// Implicitly generated code : DO NOT EDIT
FUNCTION CheckLRangeSigned : LINT
VAR_INPUT
	value, lower, upper: LINT;
END_VAR

{noflow}
IF (value < lower) THEN
	CheckLRangeSigned := lower;
	F_Log(E_LogLevel.eFatal, 'Check LINT range signed exception: {value} {lower} {upper}').WithLogger('CheckLRangeSigned').WithAnyArg(value).WithAnyArg(lower).WithAnyArg(upper).CreateLog();
ELSIF(value > upper) THEN
	CheckLRangeSigned := upper;
	F_Log(E_LogLevel.eFatal, 'Check LINT range signed exception: {value} {lower} {upper}').WithLogger('CheckLRangeSigned').WithAnyArg(value).WithAnyArg(lower).WithAnyArg(upper).CreateLog();
ELSE
	CheckLRangeSigned := value;
END_IF
{flow}

END_FUNCTION

(* stored: Version 1.1.0.1, ProductVersion 3.1.4024.0
   POU CheckLRangeSigned: Id {5e7ceb1d-2f5e-499d-8672-94a0ab371682}, SpecialFunc CheckLRangeSigned *)
